// TIA Portal V16 export
// export: Created 2021-11-12T13:33:14.6505702Z, ExportSetting WithDefaults, DisplayName Totally Integrated Automation Portal, DisplayVersion V16 Update 3, DisplayName TIA Portal Version Control Interface, DisplayVersion V16 Update 2, DisplayName TIA Portal Openness, DisplayVersion V16 Update 3, DisplayName SINAMICS Startdrive Advanced, DisplayVersion V16 Update 5, DisplayName SINAMICS Startdrive G130, G150, S120, S150, SINAMICS MV, S210, DisplayVersion V16 Update 5, DisplayName SINAMICS Startdrive G110M, G120, G120C, G120D, G120P, G115D, DisplayVersion V16 Update 5, DisplayName STEP 7 Professional, DisplayVersion V16 Update 3, DisplayName STEP 7 Safety, DisplayVersion V16, DisplayName WinCC UA Professional, DisplayVersion V16 Update 3
DATA_BLOCK "HMI_CMD_Zone400"   // DB118
{ S7_Optimized_Access := 'TRUE'; DB_Accessible_From_OPC_UA := 'FALSE' }
VERSION : 0.1
// stored: AutoNumber true, DBAccessibleFromOPCUA false, IsOnlyStoredInLoadMemory false, IsRetainMemResEnabled false, IsWriteProtectedInAS false, MemoryReserve 100
   VAR
      Mode : "UDT_Zone_Command";   // Commands for zone 400
      Station410_Mode : "UDT_Station_Command";   // Commands for station 410
      Station420_Mode : "UDT_Station_Command";   // Commands for station 420
      Station430_Mode : "UDT_Station_Command";   // Commands for station 430
      Station440_Mode : "UDT_Station_Command";   // Commands for station 440
      Station450_Mode : "UDT_Station_Command";   // Commands for station 450
      Station460_Mode { S7_SetPoint := 'True'} : "UDT_Station_Command";   // Commands for station 460
      StationTHM1_Mode { S7_SetPoint := 'True'} : "UDT_Station_Command";   // Commands for station THM1
      StationTHM2_Mode { S7_SetPoint := 'True'} : "UDT_Station_Command";   // Commands for station THM2
      StationsSum { S7_SetPoint := 'True'} : "UDT_StationsModesCmd";   // Sum of commands for stations of zone 400
   END_VAR
BEGIN
END_DATA_BLOCK
